Yaskawa INFORM job: ramp_planes_programF.JBI

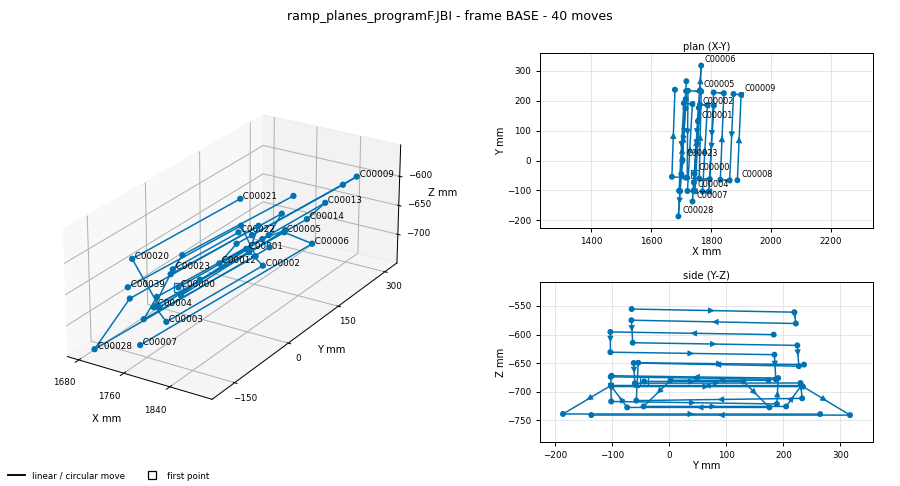
[picture p0: tool path of ramp_planes_programF.JBI in frame BASE, 40 of 46 moves have a stored position in this frame; points joined in program order, loops and branches not executed]
/JOB
//NAME ramp_planes_programF
//POS
///NPOS 40,0,40,0,0,0
///TOOL 0
///POSTYPE BASE
///RECTAN
///RCONF 0,0,0,0,0,0,0,0,0,0,0,0,0,0,0,0,0,0,0,0,0,0,0,0
C00000=1746.040607,-43.910907,-682.211692,175.000000,-89.572480,-5.000000
C00001=1757.413293,129.951574,-682.253714,175.000000,-89.572480,-5.000000
C00002=1759.979012,175.609664,-727.844933,175.000000,-89.572480,-5.000000
C00003=1743.573698,-73.823649,-727.783977,175.000000,-89.572480,-5.000000
C00004=1741.637769,-101.283923,-691.175151,180.000000,-60.000000,0.000000
C00005=1763.816463,234.265748,-691.257968,180.000000,-60.000000,0.000000
C00006=1767.731909,316.845899,-741.268230,180.000000,-60.000000,0.000000
C00007=1738.779665,-136.629916,-741.163927,180.000000,-60.000000,0.000000
C00008=1888.436048,-65.916710,-555.368102,175.000000,-46.004717,-5.000000
C00009=1900.927847,219.216482,-560.876603,175.000000,-46.004717,-5.000000
C00010=1875.644836,221.868101,-580.773298,175.000000,-46.004717,-5.000000
C00011=1862.726520,-66.386655,-574.924670,175.000000,-46.004717,-5.000000
C00012=1831.688819,-64.106483,-614.417521,175.000000,-46.004717,-5.000000
C00013=1843.382392,224.445342,-619.076482,175.000000,-46.004717,-5.000000
C00014=1809.228961,227.108185,-655.551411,175.000000,-46.004717,-5.000000
C00015=1796.499064,-62.300882,-649.911296,175.000000,-46.004717,-5.000000
C00016=1761.245587,-60.301276,-685.339067,175.000000,-46.004717,-5.000000
C00017=1767.809431,230.049224,-685.002458,175.000000,-46.004717,-5.000000
C00018=1723.782578,232.923006,-711.936940,175.000000,-46.004717,-5.000000
C00019=1720.914563,-57.826961,-715.852107,175.000000,-46.004717,-5.000000
C00020=1670.046807,-54.342751,-649.563174,180.000000,-60.000000,0.000000
C00021=1680.210027,236.159146,-652.699306,180.000000,-60.000000,0.000000
C00022=1715.468918,174.055965,-680.315766,175.000000,-88.995474,-5.000000
C00023=1705.270528,2.275534,-680.225629,175.000000,-88.995474,-5.000000
C00024=1701.477980,-45.000824,-725.991082,175.000000,-88.995474,-5.000000
C00025=1716.067875,204.836757,-726.117924,175.000000,-88.995474,-5.000000
C00026=1717.467877,231.495929,-689.533861,180.000000,-60.000000,0.000000
C00027=1697.777027,-102.213796,-689.360877,180.000000,-60.000000,0.000000
C00028=1691.750730,-186.321316,-739.306325,180.000000,-60.000000,0.000000
C00029=1718.356050,264.479699,-739.540098,180.000000,-60.000000,0.000000
C00030=1810.098538,183.080115,-600.209623,175.000000,-59.649120,-5.000000
C00031=1793.043978,-103.215575,-595.469684,175.000000,-59.649120,-5.000000
C00032=1772.252232,-103.240536,-630.997946,175.000000,-59.649120,-5.000000
C00033=1788.679159,184.352578,-635.346548,175.000000,-59.649120,-5.000000
C00034=1763.627545,186.753180,-678.581946,175.000000,-59.649120,-5.000000
C00035=1746.931590,-102.599231,-674.108039,175.000000,-59.649120,-5.000000
C00036=1721.900024,-101.745706,-717.383538,175.000000,-59.649120,-5.000000
C00037=1738.475245,188.656845,-721.767489,175.000000,-59.649120,-5.000000
C00038=1709.938546,190.919475,-676.361861,180.000000,-60.000000,0.000000
C00039=1693.851015,-101.078528,-672.292768,180.000000,-60.000000,0.000000
///POSTYPE PULSE
///PULSE
EC00000=0
EC00001=0
EC00002=0
EC00003=0
EC00004=0
EC00005=0
EC00006=0
EC00007=0
EC00008=92160
EC00009=92160
EC00010=92160
EC00011=92160
EC00012=92160
EC00013=92160
EC00014=92160
EC00015=92160
EC00016=92160
EC00017=92160
EC00018=92160
EC00019=92160
EC00020=92160
EC00021=92160
EC00022=184320
EC00023=184320
EC00024=184320
EC00025=184320
EC00026=184320
EC00027=184320
EC00028=184320
EC00029=184320
EC00030=276480
EC00031=276480
EC00032=276480
EC00033=276480
EC00034=276480
EC00035=276480
EC00036=276480
EC00037=276480
EC00038=276480
EC00039=276480
//INST
///DATE 2023/08/08 15:19
///ATTR SC,RW,RJ
////FRAME BASE
///GROUP1 RB1,ST1
NOP
MOVJ P009 EX000 VJ=15.00
MOVJ P009 VJ=15.00
MOVJ C00000 EC00000 VJ=15.0
CALL JOB:SPYON
MOVL C00001 EC00001 V=150.0
MOVL C00002 EC00002 V=150.0
MOVL C00003 EC00003 V=150.0
MOVL C00004 EC00004 V=150.0
MOVL C00005 EC00005 V=150.0
MOVL C00006 EC00006 V=150.0
MOVL C00007 EC00007 V=150.0
CALL JOB:SPYOF
MOVJ P009 VJ=15.00
MOVJ C00008 EC00008 VJ=15.0
CALL JOB:SPYON
MOVL C00009 EC00009 V=150.0
MOVL C00010 EC00010 V=150.0
MOVL C00011 EC00011 V=150.0
MOVL C00012 EC00012 V=150.0
MOVL C00013 EC00013 V=150.0
MOVL C00014 EC00014 V=150.0
MOVL C00015 EC00015 V=150.0
MOVL C00016 EC00016 V=150.0
MOVL C00017 EC00017 V=150.0
MOVL C00018 EC00018 V=150.0
MOVL C00019 EC00019 V=150.0
MOVL C00020 EC00020 V=150.0
MOVL C00021 EC00021 V=150.0
CALL JOB:SPYOF
MOVJ P009 VJ=15.00
MOVJ C00022 EC00022 VJ=15.0
CALL JOB:SPYON
MOVL C00023 EC00023 V=150.0
MOVL C00024 EC00024 V=150.0
MOVL C00025 EC00025 V=150.0
MOVL C00026 EC00026 V=150.0
MOVL C00027 EC00027 V=150.0
MOVL C00028 EC00028 V=150.0
MOVL C00029 EC00029 V=150.0
CALL JOB:SPYOF
MOVJ P009 VJ=15.00
MOVJ C00030 EC00030 VJ=15.0
CALL JOB:SPYON
MOVL C00031 EC00031 V=150.0
MOVL C00032 EC00032 V=150.0
MOVL C00033 EC00033 V=150.0
MOVL C00034 EC00034 V=150.0
MOVL C00035 EC00035 V=150.0
MOVL C00036 EC00036 V=150.0
MOVL C00037 EC00037 V=150.0
MOVL C00038 EC00038 V=150.0
MOVL C00039 EC00039 V=150.0
CALL JOB:SPYOF
MOVJ P009 VJ=15.00
END
